TYPE CyclicPos_CMD_typ :
STRUCT
	
	Start 		: BOOL;
	Disable 	: BOOL;
	
END_STRUCT
END_TYPE

(* stored: Version 1.1.0.1, ProductVersion 3.1.4024.3
   DUT CyclicPos_CMD_typ: Id {f571c72b-8786-0401-145f-77a6e93552cc} *)
